TYPE ST_Euchner_MSM_HW_OUT :
STRUCT
	///Hardware Out
	nByte0: USINT;
END_STRUCT
END_TYPE

(* stored: Version 1.1.0.1, ProductVersion 3.1.4024.12
   DUT ST_Euchner_MSM_HW_OUT: Id {c6aa8cfa-c729-4006-bd4f-3eed8edc74b8} *)
